PROGRAM MAIN
VAR
	fRand1 	: DRAND;
	iSeed 	: INT := 13;
	fTest 	: REAL;
END_VAR

fRand1(Seed:=iSeed);
sampleADSGVL.fCCATempSupPrimADS := fRand1.Num * 50.0;
sampleADSGVL.fCCATempSupADS 	:= fRand1.Num * 30.0;
sampleADSGVL.fCCATempRetADS 	:= fRand1.Num * 25.0;
sampleADSGVL.fCCATempRetPrimADS := fRand1.Num * 25.0;

END_PROGRAM

(* stored: Version 1.1.0.1, ProductVersion 3.1.4024.4
   POU MAIN: Id {38c85d5e-1444-4b25-93ab-b80f636cf0cf}, SpecialFunc None *)
